// TIA Portal project "proximi 1" (V16)

(* hardware
DEVICE "S7-1200 station_1"  S7-1200 Station
   slot 0: "Rack_0"  S7-1200 Rack  Rack  V1.0
   slot 1: "PLC_1"  CPU 1212C AC/DC/Rly  6ES7 212-1BE40-0XB0  V4.0
*)

// ===== PLC "PLC_1"  CPU 1212C AC/DC/Rly =====

VAR_GLOBAL   // PLC tag table "Default tag table"
   "start" AT %I0.0 : Bool;
   "stop" AT %I0.1 : Bool;
   "prox" AT %I0.2 : Bool;
   "km1" AT %Q0.0 : Bool;
   "km2" AT %Q0.1 : Bool;
   "km3" AT %Q0.2 : Bool;
   "Tag_1" AT %M0.0 : Bool;
   "Tag_2" AT %M1.0 : Bool;
END_VAR

// folder: System blocks/Program resources

DATA_BLOCK "T1"   // DB1
{ S7_Optimized_Access := 'TRUE' }
AUTHOR : Simatic
FAMILY : IEC
NAME : IEC_TMR
VERSION : 1.0
// stored: InstanceOfName IEC_TIMER
"IEC_TIMER"
BEGIN
END_DATA_BLOCK

// folder: (top level)

ORGANIZATION_BLOCK "Main"   // OB1, LAD, ProgramCycle
TITLE = "Main Program Sweep (Cycle)"
{ S7_Optimized_Access := 'TRUE' }
VERSION : 0.1
   VAR_INPUT
      Initial_Call : Bool;   // Initial call of this OB
      Remanence : Bool;   // =True, if remanent data are available
   END_VAR
   VAR_TEMP   // added for the SCL form of the ladder/FBD networks
      _w1 : Bool;
   END_VAR
BEGIN

REGION Network 1
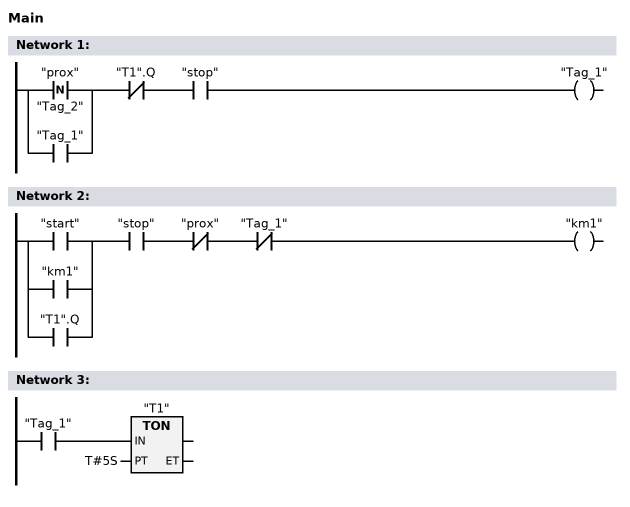
   RUNG wire#powerrail
      N_Contact(operand := "prox", bit := "Tag_2")
      wire#w1
      I_Contact( "T1".Q )
      Contact( "stop" )
      Coil( "Tag_1" )
   END_RUNG
   RUNG wire#powerrail
      Contact( "Tag_1" )
   END_RUNG wire#w1
   // the same network as SCL:
   #_w1 := NOT "prox" AND "Tag_2";   // falling edge of "prox"
   "Tag_2" := "prox";
   "Tag_1" := (#_w1 OR "Tag_1") AND NOT "T1".Q AND "stop";
END_REGION

REGION Network 2
   RUNG wire#powerrail
      Contact( "start" )
      wire#w1
      Contact( "stop" )
      I_Contact( "prox" )
      I_Contact( "Tag_1" )
      Coil( "km1" )
   END_RUNG
   RUNG wire#powerrail
      Contact( "km1" )
   END_RUNG wire#w1
   RUNG wire#powerrail
      Contact( "T1".Q )
   END_RUNG wire#w1
   // the same network as SCL:
   "km1" := ("start" OR "km1" OR "T1".Q) AND "stop" AND NOT "prox" AND NOT "Tag_1";
END_REGION

REGION Network 3
   "T1".TON(IN := "Tag_1", PT := T#5S);
END_REGION
END_ORGANIZATION_BLOCK